// TIA Portal V20 export
TYPE "LBP_typeAxisX"
TITLE = Axis interface / Interface d'axe
// User data type for blocks LBP_Axis1 [DB31] .. LBP_Axis31 [DB61] / Type de données utilisateur pour les blocs LBP_Axis1 [DB31] .. LBP_Axis31 [DB61]
   STRUCT
      A_FD_OR : Byte;   // Feedrate override / Correction d'avance
      A_DriveEnable : Bool;   // Drive test movement enable / Débloquer le déplacement pour test d'entraînement
      A_AckFixedStop : Bool;   // Acknowledge fixed stop reached / Acquittement accostage de butée
      A_SensorFixedStop : Bool;   // Sensor fixed stop / Détecteur butée
      A_ASpDisable : Bool;   // Axis/spindle disable / Désactiver axe/broche
      A_Follow_upMode : Bool;   // Follow-up mode / Mode poursuite
      A_PosMeas1 : Bool;   // Position measuring system 1 / Système de mesure de position 1
      A_PosMeas2 : Bool;   // Position measuring system 2 / Système de mesure de position 2
      A_ORactive : Bool;   // Override active / Correction active
      A_SWCam : Bool;   // SW cam activation / Activation came logicielle
      A_ContrEnable : Bool;   // Controller enable / Activer la commande
      A_DelDTGSpReset : Bool;   // Delete distance to go/Spindle-Reset / Effacer la distance restante à parcourir / Reset broche
      A_Clamp : Bool;   // Clamping in progress / Serrage en cours
      A_RefVal1 : Bool;   // Reference point value 1 / Valeur de point de référence 1
      A_RefVal2 : Bool;   // Reference point value 2 / Valeur de point de référence 2
      A_RefVal3 : Bool;   // Reference point value 3 / Valeur de point de référence 3
      A_RefVal4 : Bool;   // Reference point value 4 / Valeur de point de référence 4
      A_ExtZO : Bool;   // Import external ZO / Importer ZO externes
      A_EnabTravFixedStop : Bool;   // Enable travel to fixed stop / Activer déplacement pour accostage de butée
      A_FixedFD1 : Bool;   // Activate fixed feedrate 1 / Activer l'avance fixe 1
      A_FixedFD2 : Bool;   // Activate fixed feedrate 2 / Activer l'avance fixe 2
      A_FixedFD3 : Bool;   // Activate fixed feedrate 3 / Activer l'avance fixe 3
      A_FixedFD4 : Bool;   // Activate fixed feedrate 4 / Activer l'avance fixe 4
      A_VelocSpeedLimit : Bool;   // Velocity/spindle speed limitation / Limitation vitesse / vitesse de broche
      A_PrgtestAxRel : Bool;   // Program test axis/spindle release / Débloquer test de programme axe/broche
      A_HW1 : Bool;   // Activate handwheel 1 / Activer manivelle 1
      A_HW2 : Bool;   // Activate handwheel 2 / Activer manivelle 2
      A_HW3 : Bool;   // Activate handwheel 3 / Activer manivelle 3
      A_FDSpStop : Bool;   // Feed stop/spindle stop / Arrêt avance / arrêt broche
      A_Disable : Bool;   // Traversing key disable / Désactiver la touche de déplacement
      A_RapidTrOR : Bool;   // Rapid traverse override / Correction marche rapide
      A_Minus : Bool;   // Traversing key minus / Touche de déplacement moins
      A_Plus : Bool;   // Traversing key plus / Touche de déplacement plus
      A_INC1 : Bool;   // INC1
      A_INC10 : Bool;   // INC10
      A_INC100 : Bool;   // INC100
      A_INC1000 : Bool;   // INC1000
      A_INC10000 : Bool;   // INC10000
      A_INCVar : Bool;   // INC variable / Variable INC
      A_ContManTravel : Bool;   // Continuous manual travel / Mode manuel continu
      f5_7 : Bool;
      A_OEMAxis : Byte;   // OEM axis signals / Signaux des axes OEM
      A_InvHWDirOfRot : Bool;   // Inverting handwheel direction of rotation / Inverser sens de rotation manivelle
      f7_1 : Bool;
      f7_2 : Bool;
      f7_3 : Bool;
      f7_4 : Bool;
      f7_5 : Bool;
      f7_6 : Bool;
      f7_7 : Bool;
      A_NCASpChanA : Bool;   // Assign NC axis/spindle channel A / Affecter axe/broche CN au canal A
      A_NCASpChanB : Bool;   // Assign NC axis/spindle channel B / Affecter axe/broche CN au canal B
      A_NCASpChanC : Bool;   // Assign NC axis/spindle channel C / Affecter axe/broche CN au canal C
      A_NCASpChanD : Bool;   // Assign NC axis/spindle channel D / Affecter axe/broche CN au canal D
      A_NCASpStrobe : Bool;   // Activation of assignment with pos. edge / Activation de l'affection sur font montant
      f8_5 : Bool;
      f8_6 : Bool;
      A_PLCASp : Bool;   // Request PLC axis/spindle / Demander axe/broche AP
      A_Para_A : Bool;   // Parameter block servo A / Bloc de paramètres servo A
      A_Para_B : Bool;   // Parameter block servo B / Bloc de paramètres servo B
      A_Para_C : Bool;   // Parameter block servo C / Bloc de paramètres servo C
      A_LockParSetDef : Bool;   // Lock parameter set definition from NC / Bloquer la définition de jeu de paramètre depuis CN
      f9_4 : Bool;
      f9_5 : Bool;
      f9_6 : Bool;
      f9_7 : Bool;
      A_REPOSDelay : Bool;   // REPOS DELAY
      f10_1 : Bool;
      f10_2 : Bool;
      f10_3 : Bool;
      f10_4 : Bool;
      f10_5 : Bool;
      f10_6 : Bool;
      f10_7 : Bool;
      A_StartBrakeTest : Bool;   // Start brake test / Démarrer test de frein
      f11_1 : Bool;
      f11_2 : Bool;
      f11_3 : Bool;
      f11_4 : Bool;
      f11_5 : Bool;
      f11_6 : Bool;
      f11_7 : Bool;
      A_HWLimitMinus : Bool;   // Hardware limit switch minus / Fin de course matériel moins
      A_HWLimitPlus : Bool;   // Hardware limit switch plus / Fin de course matériel plus
      A_SWLimit2Minus : Bool;   // 2nd software limit switch minus / 2e fin de course logiciel moins
      A_SWLimit2Plus : Bool;   // 2nd software limit switch plus / 2e fin de course logiciel plus
      A_ModuloLimitEn : Bool;   // Modulo limit enabled / Limite modulo activée
      f12_5 : Bool;
      f12_6 : Bool;
      A_DelayRef : Bool;   // Delay reference point approach / Retarder l'accostage de point de référence
      A_JogFixPPos0 : Bool;   // JogFixPointPos 0
      A_JogFixPPos1 : Bool;   // JogFixPointPos 1
      A_JogFixPPos2 : Bool;   // JogFixPointPos 2
      A_JogToPos : Bool;   // Jog to position / Mode JOG vers position
      f13_4 : Bool;
      f13_5 : Bool;
      f13_6 : Bool;
      f13_7 : Bool;
      A_ProgtestSuppress : Bool;   // Program test to suppress / Inhiber test de programme
      A_ProgtestActivate : Bool;   // Activate program test / Activer test de programme
      f14_2 : Bool;
      f14_3 : Bool;
      f14_4 : Bool;
      f14_5 : Bool;
      f14_6 : Bool;
      f14_7 : Bool;
      f15 : Byte;
      A_ActGearA : Bool;   // Current gear stage A / Rapport de transmission actuel A
      A_ActGearB : Bool;   // Current gear stage B / Rapport de transmission actuel B
      A_ActGearC : Bool;   // Current gear stage C / Rapport de transmission actuel C
      A_GearChangeOv : Bool;   // Gear has changed over / Réducteur a changé de rapport
      A_Sp1Syn : Bool;   // Re-synchronize spindle 1 / Resynchroniser broche 1
      A_Sp2Syn : Bool;   // Re-synchronize spindle 2 / Resynchroniser broche 2
      A_NoMonitorGear : Bool;   // No monitoring when changing gear / Aucune surveillance pendant le changement de rapport de réducteur
      A_DeleteS : Bool;   // Delete S value / Supprimer la valeur S
      A_FD_ORSp : Bool;   // Feedrate override for spindle valid / Correction d'avance pour broche valide
      f17_1 : Bool;
      f17_2 : Bool;
      f17_3 : Bool;
      A_Sp1SynP : Bool;   // Re-synchronize spindle 1 for positioning / Resynchroniser broche 1 pour positionnement
      A_Sp2SynP : Bool;   // Re-synchronize spindle 2 for positioning / Resynchroniser broche 2 pour positionnement
      A_M3M4Inv : Bool;   // Invert M3/M4 / Inverser M3/M4
      f17_7 : Bool;
      f18_0 : Bool;
      f18_1 : Bool;
      f18_2 : Bool;
      f18_3 : Bool;
      A_OscilPLC : Bool;   // Oscillation via PLC / Oscillation via AP
      A_OscilSpeed : Bool;   // Enable Oscillation / Activer oscillation
      A_SetRotDirectRight : Bool;   // Setpoint osci. direct. right / Consigne sens d'oscillation à droite
      A_SetRotDirectLeft : Bool;   // Setpoint osci. direct. left / Consigne sens d'oscillation à gauche
      A_SpOR : Byte;   // Spindle override / Correction broche
      f20_0 : Bool;
      A_RUEncQuStop : Bool;   // Run-up encoder quick stop / Générateur de rampe Arrêt rapide
      f20_2 : Bool;
      A_SpeedSetpSmooth : Bool;   // Speed setpoint smoothing / Lissage consigne de vitesse
      f20_4 : Bool;
      A_HoldBrakeToOpen : Bool;   // Holding brake open / Frein à l'arrêt desserré
      f20_6 : Bool;
      f20_7 : Bool;
      A_ParA : Bool;   // Parameter set selection A / Jeux de paramètres sélection A
      A_ParB : Bool;   // Parameter set selection B / Jeux de paramètres sélection B
      A_ParC : Bool;   // Parameter set selection C / Jeux de paramètres sélection C
      A_MotA : Bool;   // Motor selection A / Sélection moteur A
      A_MotB : Bool;   // Motor selection B / Sélection moteur B
      A_MotOK : Bool;   // Motor selected / Moteur sélectionné
      A_IntegratDisable : Bool;   // N controller integrator disable / Commande N Désactiver intégrateur
      A_PulseEnable : Bool;   // Pulse enable / Activer impulsions
      f22_0 : Bool;
      f22_1 : Bool;
      f22_2 : Bool;
      f22_3 : Bool;
      f22_4 : Bool;
      f22_5 : Bool;
      f22_6 : Bool;
      f22_7 : Bool;
      f23_0 : Bool;
      f23_1 : Bool;
      f23_2 : Bool;
      f23_3 : Bool;
      f23_4 : Bool;
      f23_5 : Bool;
      f23_6 : Bool;
      f23_7 : Bool;
      f24_0 : Bool;
      A_ControlAx : Bool;   // Control Axis / Axe pilote
      f24_2 : Bool;
      f24_3 : Bool;
      A_TorqComp : Bool;   // Torque compensation / Compensation de couple
      A_ChangSetpOutAss0 : Bool;   // Bit value for CTRLOUT_changed - Change setpoint output assignment / Valeur de bit pour CTRLOUT_changed - Modifier l'affectation de la sortie de consigne
      A_ChangSetpOutAss1 : Bool;   // Bit value for CTRLOUT_changed - Change setpoint output assignment / Valeur de bit pour CTRLOUT_changed - Modifier l'affectation de la sortie de consigne
      A_MS : Bool;   // Main/Sub: activate coupling / Maître/esclave : activer le couplage
      A_DynBComp : Bool;   // Dynamic backlash compensation activated / Compensation dynamique de jeu activée
      f25_1 : Bool;
      f25_2 : Bool;
      f25_3 : Bool;
      f25_4 : Bool;
      f25_5 : Bool;
      f25_6 : Bool;
      f25_7 : Bool;
      f26_0 : Bool;
      f26_1 : Bool;
      f26_2 : Bool;
      A_CompContr : Bool;   // Compensation controller On / Contrôleur de compensation MARCHE
      A_FollowAxOv : Bool;   // Enable following axis override / Activer la correction de l'axe asservi
      f26_5 : Bool;
      f26_6 : Bool;
      f26_7 : Bool;
      A_DEPMCS : Bool;   // Resume: DEPMCS / Continuer : DEPMCS
      A_DEPBCS : Bool;   // Resume: DEPBCS / Continuer : DEPBCS
      A_Corr : Bool;   // Resume: Corr / Continuer : corr
      A_HIAxMove : Bool;   // Resume: HIAxMove / Continuer : HIAxMove
      A_StopDEPMCS : Bool;   // Stop: DEPMCS / Arrêt : DEPMCS
      A_StopDEPBCS : Bool;   // Stop: DEPBCS / Arrêt : DEPBCS
      A_StopCorr : Bool;   // Stop: Corr / Arrêt : corr
      A_StopHIAxMove : Bool;   // Stop: HIAxMove / Arrêt : HIAxMove
      A_OscillAxExtRev : Bool;   // OscillAxExtReversal
      A_AxReset : Bool;   // AXRESET
      A_AxResume : Bool;   // AXRESUME
      A_SetRP : Bool;   // Set reversal point / Définir point d'inversion
      A_ChangeRP : Bool;   // Change reversal point / Modifier le point d'inversion
      A_StopRP : Bool;   // Stop at next reversal point / Arrêt sur point d'inversion suivant
      A_Stop : Bool;   // Stop / Arrêt
      A_PLCAxis : Bool;   // PLC checks axis / AP vérifie axe
      f29_0 : Bool;
      f29_1 : Bool;
      f29_2 : Bool;
      f29_3 : Bool;
      A_StartGantSynRun : Bool;   // Start gantry synchronization run / Démarrer l'opération de synchronisation Gantry
      A_NoAutoSync : Bool;   // No auto sync / Aucune sync auto
      f29_6 : Bool;
      f29_7 : Bool;
      A_StopSpindle : Bool;   // Stop spindle / Arrêt broche
      A_StartCW : Bool;   // Start spindle clockwise / Démarrer broche avec rotation horaire
      A_StartCCW : Bool;   // Start spindle counterclockwise / Démarrer broche avec rotation antihoraire
      A_AutoGearStep : Bool;   // Autom. gear step change / Chmnt. auto rapport transmission
      A_PosSpindle : Bool;   // Position spindle / Position de broche
      f30_5 : Bool;
      f30_6 : Bool;
      f30_7 : Bool;
      f31_0 : Bool;
      f31_1 : Bool;
      f31_2 : Bool;
      f31_3 : Bool;
      A_Resynchronize : Bool;   // Resynchronize / Resynchroniser
      A_DisSync : Bool;   // Disable synchronization / Désactiver la synchronisation
      A_Tracksync : Bool;   // Track synchronism / Tracer synchronisme
      A_DelSyncRunCorr : Bool;   // Deleting synchronous run correction / Suppression de la correction marche synchrone
      f32_0 : Bool;
      f32_1 : Bool;
      f32_2 : Bool;
      f32_3 : Bool;
      f32_4 : Bool;
      f32_5 : Bool;
      f32_6 : Bool;
      f32_7 : Bool;
      f33_0 : Bool;
      f33_1 : Bool;
      f33_2 : Bool;
      f33_3 : Bool;
      f33_4 : Bool;
      f33_5 : Bool;
      f33_6 : Bool;
      f33_7 : Bool;
      A_SI_SetpLimBit0 : Bool;   // Set point limitation Bit0 / Limitation de consigne Bit 0
      A_SI_SetpLimBit1 : Bool;   // Set point limitation Bit1 / Limitation de consigne Bit 1
      f34_2 : Bool;
      A_ActivateBrakeRampForSs2e : Bool;   // Brakes with NCK ramp on selection of SS2E (MD36959 MA_SAFE_BRAKE_RAMP_TIME) / Freinage avec rampe du NCK lors de la sélection de SS2E (MD36959 MA_SAFE_BRAKE_RAMP_TIME)
      f34_4 : Bool;
      f34_5 : Bool;
      f34_6 : Bool;
      f34_7 : Bool;
      f35 : Byte;
      f36 : Array[36..55] of Byte;
      A_FeedDriveCAxEng : Bool;   // Separate feed drive as C axis engaged / Entraînement d'avance séparé activé en tant qu'axe C
      A_SpSpeedDisp : Bool;   // Spindle speed display / Affichage vitesse de broche
      A_SpInsideClamp : Bool;   // Spindle inside clamping / Serrage interne broche
      f56_3 : Bool;
      f56_4 : Bool;
      f56_5 : Bool;
      f56_6 : Bool;
      f56_7 : Bool;
      f57 : Byte;
      f58 : Word;
      E_SpNA : Bool;   // Spindle/no axis / Broche / aucun axe
      E_NCU_Link : Bool;   // NCU_link active axis / NCU_link axe actif
      E_EncodFreq1 : Bool;   // Encoder limit frequency 1 exceeded / Fréquence limite capteur 1 dépassée
      E_EncodFreq2 : Bool;   // Encoder limit frequency 2 exceeded / Fréquence limite capteur 2 dépassée
      E_RefSyn1 : Bool;   // Referenced/synchronized 1 / Référencé/synchronisé 1
      E_RefSyn2 : Bool;   // Referenced/synchronized 2 / Référencé/synchronisé 2
      E_ExactCoarse : Bool;   // Position reached with exact stop coarse / Position atteinte avec arrêt précis approx.
      E_ExactFine : Bool;   // Position reached with exact stop fine / Position atteinte avec arrêt précis fin
      E_TravRequ : Bool;   // Travel request / Demande de déplacement
      E_AxialAlarm : Bool;   // Axial alarm / Alarme d'axe
      E_AxisReady : Bool;   // Axis ready / Axe prêt
      E_Follow_upMode : Bool;   // Follow-up mode active / Mode poursuite actif
      E_Stat : Bool;   // Axis/spindle stationary (n<nmin) / Axe/broche à l'arrêt (n<nmin)
      E_PositContr : Bool;   // Position controller active / Commande de positionnement active
      E_SpeedContr : Bool;   // Speed controller active / Régulateur de vitesse actif
      E_CurrentContr : Bool;   // Current controller active / Commande actuelle active
      E_SWCam : Bool;   // Software cams active / Came logicielle active
      E_HWOverlay : Bool;   // Handwheel overlay active / Superposition manivelle actif
      E_RevFD : Bool;   // Revolutional feedrate active / Avance par tour active
      E_MeasAct : Bool;   // Measuring active / Mesurage actif
      E_ActTravFStop : Bool;   // Activate travel to fixed stop / Activer déplacement pour accostage de butée
      E_FixedStop : Bool;   // Fixed stop reached / Butée atteinte
      E_ForceFixedStop : Bool;   // Force fixed stop limited / Force butée limitée
      E_AxContainerRot : Bool;   // Axis container rotation active / Conteneur d'axe Rotation activée
      E_AxReset : Bool;   // Axis reset done / Reset axe effectué
      E_PLCCtrlAx : Bool;   // PLC controlled axis / Axe commandé par AP
      E_AxStop : Bool;   // Axis stop active / Arrêt d'axe actif
      E_AxSpDisable : Bool;   // Axis/spindle disable active / Désactivation axe/broche active
      E_StopDEPMCS : Bool;   // Stop DEPMCS active / Arrêt DEPMCS actif
      E_StopDEPBCS : Bool;   // Stop DEPBCS active / Arrêt DEPBCS actif
      E_StopCorr : Bool;   // Stop Corr active / Arrêt corr actif
      E_StopHIAxMove : Bool;   // Stop HIAxMove active / Arrêt HIAxMove actif
      E_HW1 : Bool;   // Handwheel 1 active / Manivelle 1 active
      E_HW2 : Bool;   // Handwheel 2 active / Manivelle 2 active
      E_HW3 : Bool;   // Handwheel 3 active / Manivelle 3 active
      f64_3 : Bool;
      E_TReqMinus : Bool;   // Travel request minus / Demande de déplacement moins
      E_TReqPlus : Bool;   // Travel request plus / Demande de déplacement plus
      E_TCMinus : Bool;   // Traverse command minus / Instruction de déplacement moins
      E_TCPlus : Bool;   // Traverse command plus / Instruction de déplacement plus
      E_INC1 : Bool;   // INC1
      E_INC10 : Bool;   // INC10
      E_INC100 : Bool;   // INC100
      E_INC1000 : Bool;   // INC1000
      E_INC10000 : Bool;   // INC10000
      E_INCVar : Bool;   // INC variable / Variable INC
      E_ContManTravelAct : Bool;   // Continuous manual travel active / Mode manuel continu actif
      f65_7 : Bool;
      E_OEMAxis : Byte;   // OEM axis signals / Signaux des axes OEM
      E_InvHWDirOfRot : Bool;   // Handwheel direction of rotation invert actively / Inverser activement sens manivelle
      f67_1 : Bool;
      f67_2 : Bool;
      f67_3 : Bool;
      f67_4 : Bool;
      f67_5 : Bool;
      f67_6 : Bool;
      f67_7 : Bool;
      E_NCASpChanA : Bool;   // NC axis/spindle in channel A / Axe/broche CN dans canal A
      E_NCASpChanB : Bool;   // NC axis/spindle in channel B / Axe/broche CN dans canal B
      E_NCASpChanC : Bool;   // NC axis/spindle in channel C / Axe/broche CN dans canal C
      E_NCASpChanD : Bool;   // NC axis/spindle in channel D / Axe/broche CN dans canal D
      E_PLCType : Bool;   // New type requested by PLC / Nouveau type demandé de l'AP
      E_ChPoss : Bool;   // Change axis possible / Modification d'axe possible
      E_NeutrASp : Bool;   // Neutral axis/spindle / Axe/broche neutre
      E_PLCASp : Bool;   // PLC axis/spindle / Axe/broche AP
      E_ParS_A : Bool;   // Parameter block servo A / Bloc de paramètres servo A
      E_ParS_B : Bool;   // Parameter block servo B / Bloc de paramètres servo B
      E_ParS_C : Bool;   // Parameter block servo C / Bloc de paramètres servo C
      E_NCUNumLink_3 : Bool;
      E_NCUNumLink_4 : Bool;
      E_NCUNumLink_5 : Bool;
      E_NCUNumLink_6 : Bool;
      E_NCUNumLink_7 : Bool;
      E_ReposSh : Bool;   // REPOS shift / REPOS Décalage
      E_ReposShValid : Bool;   // REPOS shift valid / REPOS Décalage valide
      E_ReposDelayQuit : Bool;   // REPOS delay quit / REPOS Terminer temporisation
      f70_3 : Bool;
      f70_4 : Bool;
      E_SI_Drv_SICSCC : Bool;   // DRV-Safety Integrated with SIC/SCC active / DRV Safety Integrated avec SIC/SCC actif
      E_SI_Drv_Parameterized : Bool;   // Drive based Safety Intergated (SI) function enabled (at least one function in parameter "p9501" or "p9601" is parameterized) / Fonction Drive based Safety Integrated (SI) débloquée (au moins une fonction est paramétrée dans le paramètre "p9501" ou "p9601")
      f70_7 : Bool;
      E_BrakeTest : Bool;   // Brake test active / Test de frein actif
      f71_1 : Bool;
      f71_2 : Bool;
      f71_3 : Bool;
      E_POS_RESTORED1 : Bool;   // POS_RESTORED 1
      E_POS_RESTORED2 : Bool;   // POS_RESTORED 2
      f71_6 : Bool;
      E_PLCAxDedic : Bool;   // PLC axis dedicated / Axe AP dédié
      E_MMC_REPOSDelay : Bool;   // HMI REPOS DELAY
      f72_1 : Bool;
      f72_2 : Bool;
      f72_3 : Bool;
      f72_4 : Bool;
      f72_5 : Bool;
      f72_6 : Bool;
      f72_7 : Bool;
      f73 : Byte;
      f74_0 : Bool;
      f74_1 : Bool;
      f74_2 : Bool;
      f74_3 : Bool;
      E_ModLimEnAct : Bool;   // Modulo limit enabled active / Limite modulo activée actif
      f74_5 : Bool;
      f74_6 : Bool;
      f74_7 : Bool;
      E_JogFixPPos0Act : Bool;   // JogFixPointPos 0 active / JogFixPointPos 0 activé
      E_JogFixPPos1Act : Bool;   // JogFixPointPos 1 active / JogFixPointPos 1 activé
      E_JogFixPPos2Act : Bool;   // JogFixPointPos 2 active / JogFixPointPos 2 activé
      E_JogFixPPos0 : Bool;   // JogFixPointPos 0 reached / JogFixPointPos 0 atteint
      E_JogFixPPos1 : Bool;   // JogFixPointPos 1 reached / JogFixPointPos 1 atteint
      E_JogFixPPos2 : Bool;   // JogFixPointPos 2 reached / JogFixPointPos 2 atteint
      E_JogToPos : Bool;   // Jog to position active / Mode JOG vers position actif
      E_JogPos : Bool;   // Jog position reached / Position JOG atteinte
      E_ScratchPulse : Bool;   // Scratch pulse
      f76_1 : Bool;
      f76_2 : Bool;
      f76_3 : Bool;
      E_PathAxis : Bool;   // Path axis / Axe d'interpolation
      E_PosAxis : Bool;   // Positioning axis / Axe de positionnement
      E_IndexAxisPos : Bool;   // Indexing axis in position / Axe indexé en position
      E_CurvePos : Bool;   // Curve axis in position / Axe de contournage en position
      E_CollCheckRedSpeed : Bool;   // Reduced speed of Collisions Check / Vitesse réduite du contrôle de collision
      f77_1 : Bool;
      f77_2 : Bool;
      f77_3 : Bool;
      f77_4 : Bool;
      f77_5 : Bool;
      f77_6 : Bool;
      f77_7 : Bool;
      E_FPosAxis : Real;   // F function (REAL format) for positioning axes / Fonction F (format REAL) pour axes de positionnement
      E_SetpGearA : Bool;   // Setpoint gear stage A / Consigne de rapport de transmission A
      E_SetpGearB : Bool;   // Setpoint gear stage B / Consigne de rapport de transmission B
      E_SetpGearC : Bool;   // Setpoint gear stage C / Consigne de rapport de transmission C
      E_GearChange : Bool;   // Gear changeover / Changement de rapport réducteur
      f82_4 : Bool;
      f82_5 : Bool;
      f82_6 : Bool;
      f82_7 : Bool;
      E_SpeedLimit : Bool;   // Speed limit exceeded / Limite de vitesse dépassée
      E_SetSpeedLimit : Bool;   // Setpoint speed limited / Consigne de vitesse limitée
      E_SetSpeedIncreased : Bool;   // Setpoint speed increased / Consigne de vitesse augmentée
      E_GeoMonit : Bool;   // Geometry monitoring / Surveillance de géométrie
      E_SupportAreaViol : Bool;   // Support area limits violated / Limites de la zone de support dépassées
      E_SetRange : Bool;   // Spindle in setpoint range / Broche dans la plage consigne
      E_SpeedMonit : Bool;   // Speed monitoring / Surveillance de vitesse
      E_ActRotRight : Bool;   // Actual rotation direction right / Sens de rotation actuel horaire
      E_ConstCuttSpeed : Bool;   // Const. cutting speed active / Vitesse de coupe constante active
      E_SUG : Bool;   // SUG active (grinding wheel surface speed) / VPM active (vitesse périphérique de meule)
      E_CLG : Bool;   // CLG active / CLG actif
      E_Tapping : Bool;   // Tapping without compensating chuck / Taraudage sans porte-taraud compensateur
      E_SyncMode : Bool;   // Synchronous mode spindle active / Mode broche synchrone actif
      E_PosMode : Bool;   // Positioning mode spindle active / Mode positionnement broche actif
      E_OscillMode : Bool;   // Oscillation mode spindle active / Mode oscillation broche actif
      E_ContrMode : Bool;   // Control mode spindle active / Mode de commande broche actif
      E_ToolDynLimit : Bool;   // Tool with dynamics limit / Outil avec limite dynamique
      f85_1 : Bool;
      f85_2 : Bool;
      f85_3 : Bool;
      f85_4 : Bool;
      E_SpInPosition : Bool;   // Spindle in position / Broche en position
      f85_6 : Bool;
      f85_7 : Bool;
      E_MFunct : Int;   // M function (INT) for spindle / Fonction M (INT) pour broche
      E_SFunct : Real;   // S function (REAL) for spindle / Fonction S (REAL) pour broche
      f92_0 : Bool;
      E_RUEncDisabl : Bool;   // Run-up encoder disable active / Blocage codeur de démarrage actif
      f92_2 : Bool;
      E_SpeedSetpSmooth : Bool;   // Speed setpoint smoothing active / Lissage consigne de vitesse actif
      E_RLIact : Bool;   // RLI active / RLI actif
      E_HoldBrakeOpened : Bool;   // Holding brake opened / Frein à l'arrêt desserré
      f92_6 : Bool;
      E_DriveRunEn : Bool;   // Drive run enabled / Déplacement entraînement activé
      E_ParA : Bool;   // Active parameter set A / Jeux de paramètres actif A
      E_ParB : Bool;   // Active parameter set B / Jeux de paramètres actif B
      E_ParC : Bool;   // Active parameter set C / Jeux de paramètres actif C
      E_MotA : Bool;   // Active motor A / Moteur actif A
      E_MotB : Bool;   // Active motor B / Moteur actif B
      E_MotOK : Bool;   // Drive ready / Entraînement prêt
      E_IntegratDisable : Bool;   // N controller integrator disabled / Commande N Intégrateur désactivé
      E_PulseEnable : Bool;   // Pulses enabled / Impulsions débloquées
      E_MTempWarn : Bool;   // Prewarning motor temperature / Avertissement température moteur
      E_HTempWarn : Bool;   // Prewarning heat sink temperature / Avertissement température radiateur
      E_RUComplete : Bool;   // Ramp-up complete / Démarrage terminé
      E_MdMdx : Bool;   // Md<Mdx
      E_NactNmin : Bool;   // nact<nmin
      E_NactNx : Bool;   // nact<nx
      E_NactNset : Bool;   // nact=nset
      E_Message : Bool;   // Variable message function 1 / Fonction de signalisation variable 1
      E_UDClessAlThreshold : Bool;   // UDC-link < alarm threshold / Lien UDC < seuil d'alarme
      E_DcVoltageAlarmAct : Bool;   // ESR: DC link voltage is below the specified minimum / AER : la tension du circuit intermédiaire est inférieure au minimum spécifié
      E_GeneratorOperationAct : Bool;   // ESR: generator operation is active / AER : le fonctionnement du générateur est actif
      E_SpeedBelowMin : Bool;   // ESR: actual speed is below specified minimum speed - axis is a generator axis / AER : la vitesse réelle est inférieure à la vitesse minimale spécifiée – l'axe est un axe de générateur
      E_Message2 : Bool;   // Variable message function 2 / Fonction de signalisation variable 2
      E_Message3 : Bool;   // Variable message function 3 / Fonction de signalisation variable 3
      f95_6 : Bool;
      E_I2TLimit : Bool;   // Power Section I2T limit / Partie puissance limite I2T
      f96_0 : Bool;
      E_AxisCtrl : Bool;   // Axis control active / Commande d'axe active
      E_MSFine : Bool;   // Main/Sub: speed difference is within the fine tolerance range / Maître/esclave : la différence de vitesse se situe dans la plage de tolérance fine
      E_MSCoarse : Bool;   // Main/Sub: speed difference is within the coarse tolerance range / Maître/esclave : la différence de vitesse se situe dans la plage de tolérance grossière
      E_MSCompContr : Bool;   // Main/Sub: torque compensatory controller is active / Maître/esclave : le régulateur de compensation de couple est actif
      E_BitValCtrlOutChang0 : Bool;   // Bit value for CTRLOUT_changed 0: Change setpoint output assignment / Valeur de CTRLOUT_changed 0 : modifier l'affectation de sortie de consigne
      E_BitValCtrlOutChang1 : Bool;   // Bit value for CTRLOUT_changed 1: Change setpoint output assignment / Valeur de CTRLOUT_changed 1 : modifier l'affectation de sortie de consigne
      E_MS : Bool;   // Main/Sub: coupling is active / Maître/esclave : le couplage est actif
      f97 : Byte;
      E_SyncronFine : Bool;   // Synchronism fine / Synchronisme fin
      E_SyncronCoarse : Bool;   // Synchronism coarse / Synchronisme approx
      E_ActValCoupling : Bool;   // Actual value coupling / Valeur réelle couplage
      f98_3 : Bool;
      E_OverlayMotion : Bool;   // Overlaid motion / Mouvement superposé
      E_SWL : Bool;   // Speed warning limit reached / Valeur limite d'alarme pour vitesse atteinte
      E_AWL : Bool;   // Acceleration warning limit reached / Valeur limite d'alarme pour accélération atteinte
      E_EmRetr : Bool;   // Emergency retraction active / Retrait d'urgence actif
      E_MasterSp : Bool;   // Generic coupling: spindle is leading spindle / Couplage générique : la broche est une broche pilote
      E_SlaveSp : Bool;   // Generic coupling: spindle is following spindle / Couplage générique : la broche est une broche asservie
      E_SyncRunCorrDOut : Bool;   // Synchronous run correction driven out / Correction synchronisme dépassée
      E_AxisAccel : Bool;   // Axis accelerated / Axe accéléré
      E_Sync : Bool;   // Synchronization active / Synchronisation active
      E_MSR : Bool;   // Max. speed reached / Vitesse max. atteinte
      E_MAR : Bool;   // Max. acceleration reached / Accélération max. atteinte
      f99_7 : Bool;
      f100_0 : Bool;
      f100_1 : Bool;
      E_OscillAxExtRev : Bool;   // OscillAxExt Reversal active / OscillAxExt Inversion active
      E_StopOscill : Bool;   // Oscillation cannot start / Impossible de démarrer oscillation
      E_ErrorOscill : Bool;   // Error during oscillation / Erreur lors de l'oscillation
      E_SparkOut : Bool;   // Spark-out active / Passes à lécher actives
      E_OscillMotion : Bool;   // Oscillation motion active / Mouvement d'oscillation actif
      E_Oscill : Bool;   // Oscillation active
      f101_0 : Bool;
      f101_1 : Bool;
      E_GantCOLimit : Bool;   // Gantry cut-off limit exceeded / Limite coupure axe Gantry atteinte
      E_GantWarn : Bool;   // Gantry warning limit exceeded / Gantry Limite d'alarme dépassée
      E_SynRunStart : Bool;   // Synchronization run ready to start / Synchronisme prêt à démarrer
      E_GantGroupSyn : Bool;   // Gantry grouping is synchronous / Groupage Gantry synchronisé
      E_GantLeadAxis : Bool;   // Gantry leading axis / Axe pilote Gantry
      E_GantAxis : Bool;   // Gantry axis / Axe Gantry
      E_DynBComp : Bool;   // Dynamic backlash compensation activated / Compensation dynamique de jeu activée
      f102_1 : Bool;
      f102_2 : Bool;
      E_ClampTolerance : Bool;   // Clamp tolerance exceeded / Tolérance de serrage d'axe dépassée
      f102_4 : Bool;
      E_PosMeas1 : Bool;   // Position measuring system 1 active / Système de mesure de position 1 actif
      E_PosMeas2 : Bool;   // Position measuring system 2 active / Système de mesure de position 2 actif
      f102_7 : Bool;
      E_SyncRunCorrIncl : Bool;   // Synchronous run correction is included / Correction synchronisme incluse
      f103_1 : Bool;
      f103_2 : Bool;
      f103_3 : Bool;
      E_Syncron2Fine : Bool;   // Synchronism fine / Synchronisme fin
      E_Syncron2Coarse : Bool;   // Synchronism coarse / Synchronisme approx
      f103_6 : Bool;
      f103_7 : Bool;
      E_AIAxis : Array[1..31] of Bool;   // Active infeed axis[1..31] / Axe de pénétration active [1..31]
      f108_0 : Bool;
      f108_1 : Bool;
      f108_2 : Bool;
      f108_3 : Bool;
      f108_4 : Bool;
      f108_5 : Bool;
      f108_6 : Bool;
      f108_7 : Bool;
      f109_0 : Bool;
      f109_1 : Bool;
      f109_2 : Bool;
      f109_3 : Bool;
      f109_4 : Bool;
      f109_5 : Bool;
      f109_6 : Bool;
      f109_7 : Bool;
      f110_0 : Bool;
      f110_1 : Bool;
      f110_2 : Bool;
      f110_3 : Bool;
      f110_4 : Bool;
      f110_5 : Bool;
      f110_6 : Bool;
      f110_7 : Bool;
      f111_0 : Bool;
      f111_1 : Bool;
      f111_2 : Bool;
      f111_3 : Bool;
      f111_4 : Bool;
      f111_5 : Bool;
      f111_6 : Bool;
      f111_7 : Bool;
      f112 : Byte;
      f113 : Byte;
      f114 : Byte;
      f115 : Byte;
      f116 : Byte;
      f117_0 : Bool;
      f117_1 : Bool;
      f117_2 : Bool;
      f117_3 : Bool;
      f117_4 : Bool;
      f117_5 : Bool;
      f117_6 : Bool;
      f117_7 : Bool;
      f118 : DWord;
      f122 : DWord;
      f126 : Word;   // Internal / Interne
      E_MMC_ProgtestSuppress : Bool;   // HMI->PLC: Suppress program test / HMI ->AP : inhiber test de programme
      E_MMC_ProgtestActivate : Bool;   // HMI->PLC: Activate program test / HMI ->AP : activer test de programme
      f128_2 : Bool;
      f128_3 : Bool;
      f128_4 : Bool;
      f128_5 : Bool;
      f128_6 : Bool;
      f128_7 : Bool;
      f129 : Byte;
      E_FormatBit0DDS : Bool;   // Bit 0 for drive data set switchover (DDS) / Bit 0 pour la commutation du jeu de paramètres d'entraînement (DDS)
      E_FormatBit1DDS : Bool;   // Bit 1 for drive data set switchover (DDS) / Bit 1 pour la commutation du jeu de paramètres d'entraînement (DDS)
      E_FormatBit2DDS : Bool;   // Bit 2 for drive data set switchover (DDS) / Bit 2 pour la commutation du jeu de paramètres d'entraînement (DDS)
      E_FormatBit3DDS : Bool;   // Bit 3 for drive data set switchover (DDS) / Bit 3 pour la commutation du jeu de paramètres d'entraînement (DDS)
      E_FormatBit4DDS : Bool;   // Bit 4 for drive data set switchover (DDS) / Bit 4 pour la commutation du jeu de paramètres d'entraînement (DDS)
      f130_5 : Bool;
      f130_6 : Bool;
      E_MDS_DDS_InterfacesValid : Bool;   // Motor and drive data set interfaces invalid / Jeux de paramètres moteur et d'entraînement Interfaces valides
      f131 : Byte;
      E_SensorAv : Bool;   // Sensors available / Capteurs disponibles
      E_S1aMeasARod : Bool;   // Sensor S1: analogous measurement position of actuating rod / Capteur S1 : position de mesure analogique de la tige d'actionnement
      f132_2 : Bool;
      f132_3 : Bool;
      E_S4dPistonStopP : Bool;   // Sensor S4: digital value piston stop position / Capteur S4 : valeur numérique position d'arrêt piston
      E_S5dAngleShaft : Bool;   // Sensor S5: digital value angle situation shaft / Capteur S5 : valeur numérique position angulaire arbre
      E_S6Temp : Bool;   // Sensor S6: temperature / Capteur S6 : température
      f132_7 : Bool;
      f133 : Byte;
      E_ClampingState : Int;   // State of the clamping system / État du système de serrage
      E_AnalogSensor : Int;   // Analog sensor on the motor / Capteur analogique sur moteur
      f138_0 : Bool;
      f138_1 : Bool;
      f138_2 : Bool;
      f138_3 : Bool;
      E_S4PistonStopP : Bool;   // Sensor S4: piston stop position / Capteur S4 : position d'arrêt piston
      E_S5AngleShaft : Bool;   // Sensor S5: angle situation shaft / Capteur S5 : position angulaire arbre
      f138_6 : Bool;
      f138_7 : Bool;
      f139 : Byte;
      SCC : Struct   // PLC to Drive (SCC) / AP vers entraînement (SCC)
         CW1 : Struct
            TeststopStart : Bool;   // Test stops for extended functions / Stops pour test pour fonctions étendues
            res140_1 : Bool;
            res140_2 : Bool;
            res140_3 : Bool;
            res140_4 : Bool;
            CloseBrake : Bool;   // Close internal Brake / Serrer le frein interne
            res140_6 : Bool;
            res140_7 : Bool;
            res141 : Byte;
         END_STRUCT;
         CW3 : Struct
            res142 : Byte;
            SelectionSBT : Bool;   // Selection: safe brake test / Sélection : test de frein sûr
            BT_Start : Bool;   // Start: brake test / Démarrage : test de frein
            Brake_1_2 : Bool;   // Brake test with brake 1 or 2 / Test de frein avec frein 1 ou 2
            DirOfROT : Bool;   // Direction of rotation / Sens de rotation
            Testseq_1_2 : Bool;   // Test sequence 1 or 2 / Séquence de test 1 ou 2
            BrakeClosed : Bool;   // Feedback external brake / Signalisation en retour frein externe
            res143_6 : Bool;
            res143_7 : Bool;
         END_STRUCT;
      END_STRUCT;
      res144_163 : Array[144..163] of Byte;
      SIC : Struct   // Drive to PLC (SIC) / Entraînement vers AP (SIC)
         SW1 : Struct
            SLA_Sel : Bool;   // Safely Limited Acceleration selected / Accélération limitée sûre sélectionnée
            SLS_LimBit0_Sel : Bool;   // Safely-Limited Speed: limit Bit0 selected / Vitesse limitée sûre : limite bit0 sélectionnée
            SLS_LimBit1_Sel : Bool;   // Safely-Limited Speed: limit Bit1 selected / Vitesse limitée sûre : limite bit1 sélectionnée
            res164_3 : Bool;
            res164_4 : Bool;
            res164_5 : Bool;
            ESR_Req : Bool;   // Extended Stop and Retract requested / Arrêt étendu et retrait demandé
            SF_Message_Act : Bool;   // Safety error active / Erreur de sécurité active
            STO_Act : Bool;   // Safe torque off: active / Suppression sûre du couple : active
            SS1_Act : Bool;   // Safe Stop1: active / Stop sûr 1 : actif
            SS2_Act : Bool;   // Safe Stop2: active / Stop sûr 2 : actif
            SOS_Act : Bool;   // Safe Operating Stop: active / Arrêt de fonctionnement sûr : actif
            SLS_Act : Bool;   // Safely-Limited Speed: active / Vitesse limitée sûre : active
            SOS_Sel : Bool;   // Safe Operating Stop: selected / Arrêt de fonctionnement sûr : sélectionné
            SLS_Sel : Bool;   // Safely-Limited Speed: selected / Vitesse limitée sûre : sélectionnée
            InternalEvent : Bool;   // Safety error with Stop A active / Erreur de sécurité avec butée A active
         END_STRUCT;
         SW2 : Struct
            SDI_P_Sel : Bool;   // Safe direction positive: selected / Direction sûre positive : sélectionnée
            SDI_N_Sel : Bool;   // Safe direction negative: selected / Direction sûre négative : sélectionnée
            res166_2 : Bool;
            res166_3 : Bool;
            TestStopAct : Bool;   // Test stop active / Stop pour test actif
            TestStopReq : Bool;   // Test stop requested / Stop pour test demandé
            res166_6 : Bool;
            res166_7 : Bool;
            res167_0 : Bool;
            res167_1 : Bool;
            res167_2 : Bool;
            res167_3 : Bool;
            SLP_LimBit0_Sel : Bool;   // Safely-Limited Position: limit Bit0 selected / Position limitée sûre : limite bit0 sélectionnée
            res167_5 : Bool;
            res167_6 : Bool;
            SLP_Sel : Bool;   // Safely-Limited Position: selected / Position limitée sûre : sélectionnée
         END_STRUCT;
         V_Limit_B : DInt;   // Setpoint speed limit effective / Limite de consigne de vitesse active
         SW3 : Struct
            res172_0 : Bool;
            res172_1 : Bool;
            res172_2 : Bool;
            SS2E_ACTIVE : Bool;   // SS2E active / SS2E actif
            SS2ESR : Bool;   // SS2ESR active / SS2ESR actif
            res172_5 : Bool;
            AcceptSLPAct : Bool;   // Acceptance test Safely-Limited Position active / Essai de réception position limitée sûre : actif
            AcceptTestSel : Bool;   // Acceptance test selected / Essai de réception sélectionné
            SBT_Sel : Bool;   // Safety break test: selected / Test de frein de sécurité : sélectionné
            SetpSettingDrive : Bool;   // Setpoint input is in the drive during the SBT / L'entrée de consigne est dans l'entraînement pendant le SBT
            Brake_1_2 : Bool;   // Test with brake 1 or 2 / Test avec frein 1 ou 2
            BT_Act : Bool;   // Brake test: active / Test de frein : actif
            BT_OK : Bool;   // Brake test: OK / Test de frein : OK
            BT_Finished : Bool;   // Brake test: finished / Test de frein : terminé
            BrakeReq : Bool;   // External brake close requested / Serrage de frein externe demandé
            SignLoadTorque : Bool;   // Sign of load torque is negative / Signe couple de charge négatif
         END_STRUCT;
      END_STRUCT;
      res174_187 : Array[174..187] of Byte;
      CW7 : Struct
         ReservedBit08 : Bool;
         ReservedBit09 : Bool;
         ReservedBit10 : Bool;
         ReservedBit11 : Bool;
         ReservedBit12 : Bool;
         ReservedBit13 : Bool;
         ReservedBit14 : Bool;
         ReservedBit15 : Bool;
         A_DisablePowerReduction : Bool;   // DYNEGMA: disable power reduction / DYNEGMA : désactiver la réduction de puissance
         A_DisableCurrReduction : Bool;   // Motor overtemperature: disable current reduction / Surchauffe du moteur : désactiver la réduction de puissance
         ReservedBit02 : Bool;
         ReservedBit03 : Bool;
         ReservedBit04 : Bool;
         ReservedBit05 : Bool;
         ReservedBit06 : Bool;
         ReservedBit07 : Bool;
      END_STRUCT;
      SW7 : Struct
         E_EncMaintenanceRequired : Bool;   // Encoder maintenance required / Maintenance du codeur requise
         ReservedBit09 : Bool;
         ReservedBit10 : Bool;
         ReservedBit11 : Bool;
         ReservedBit12 : Bool;
         ReservedBit13 : Bool;
         ReservedBit14 : Bool;
         ReservedBit15 : Bool;
         E_TorqueLimited : Bool;   // DYNEGMA: torque limited / DYNEGMA : couple limité
         E_CurrReductionActive : Bool;   // Motor overtemperature: current reduction active / Surchauffe du moteur : réduction de puissance active
         E_MotorTempModelAlarm : Bool;   // Motor overtemperature: motor temperature model alarm active / Surchauffe du moteur : alarme de modèle thermique du moteur active
         E_PolePosIdentPassed : Bool;   // Pole position identification with encoder successfully carried out / Identification de la position des pôles avec codeur effectuée avec succès
         ReservedBit04 : Bool;
         ReservedBit05 : Bool;
         E_AndConditionFulfilled : Bool;   // AND logic operation: condition fulfilled / Opération logique ET : condition remplie
         E_OrConditionFulfilled : Bool;   // OR logic operation: condition fulfilled / Opération logique OU : condition remplie
      END_STRUCT;
   END_STRUCT;
END_TYPE
